TYPE DefrostParameters :
STRUCT
	EN: BOOL := TRUE; // $(setup)
	ENO: BOOL;
	
	T_QM1_1: BOOL;
	T_QM1_2: BOOL;
	T_QM1_3: BOOL;
	T_QM1_4: BOOL;
	T_QM1_5: BOOL;
	T_QM1_6: BOOL;
	
	Sections: INT := 4; // $(setup)
	DefrostTemperature: LREAL := -4; // $(setup)
	
	SectionTime: TIME := T#10M; // $(setup)
	
	CurrentStage: INT;
	CurrentSection: INT;
	CurrentPressureLimit: LREAL;

	DefrostState: DefrostStates;
	Stage1: DefrostStageParameters := (PressureLimit := 100, SupplyAir := 0.8, ExtractAir := 1);
	Stage2: DefrostStageParameters := (PressureLimit := 150, SupplyAir := 0.4, ExtractAir := 1);
	Stage3: DefrostStageParameters := (PressureLimit := 200, SupplyAir := 0, ExtractAir := 0.5);
	
	CurrentTime: LTIME;
	//SetPointReduction: SetPointReductionParameters;
	//ExtendedDefrost: ExtendedDefrostParameters;
	//WinterShutdown: WinterShutdownParameters;
	
END_STRUCT
END_TYPE

(* stored: Version 1.1.0.1, ProductVersion 3.1.4024.6
   DUT DefrostParameters: Id {71bafd84-79e8-4599-a31a-31f9c5bb9b99} *)
